(* PLC project Unnamed, Unknown Unnamed 1 *)
(* stored: creationDateTime 2025-11-05T11:22:18, modificationDateTime 2025-11-05T11:34:46 *)

PROGRAM main
  VAR
    Mode1SW : BOOL := False;
    Mode2SW : BOOL := False;
    Mode3SW : BOOL := False;
    Mode1 : BOOL := False;
    Mode2 : BOOL := False;
    Mode3 : BOOL := False;
    Off : BOOL := False;
  END_VAR

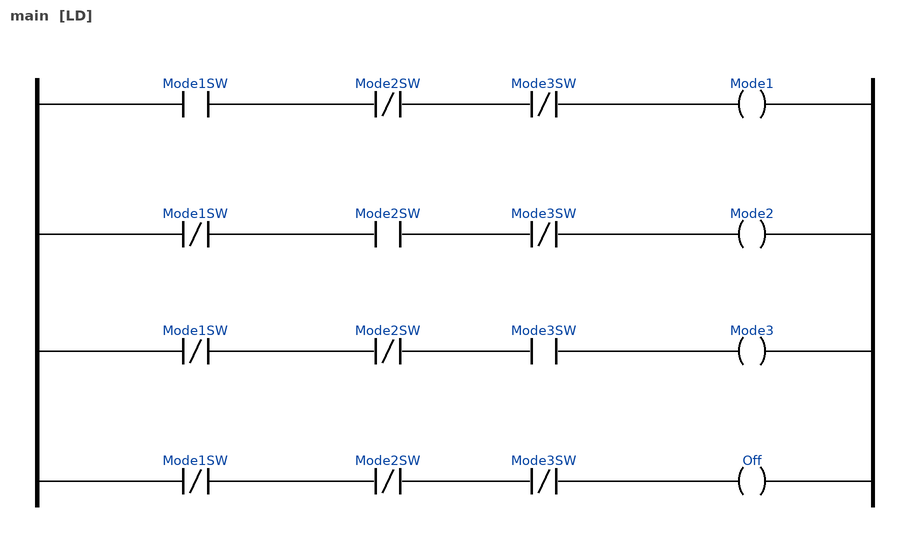
(* LD diagram, written out as Structured Text *)
Mode1 := Mode1SW AND NOT Mode2SW AND NOT Mode3SW;
Mode2 := NOT Mode1SW AND Mode2SW AND NOT Mode3SW;
Mode3 := NOT Mode1SW AND NOT Mode2SW AND Mode3SW;
Off := NOT Mode1SW AND NOT Mode2SW AND NOT Mode3SW;
END_PROGRAM

CONFIGURATION Config0
  RESOURCE Res0 ON PLC
    TASK task0(INTERVAL := T#20ms, PRIORITY := 0);
    PROGRAM instance0 WITH task0 : main;
  END_RESOURCE
END_CONFIGURATION
